PROGRAM MAIN
VAR
	SpeedMotor: MotorVarSpeed_FB;
END_VAR

SpeedMotor(
	Run:= , 
	Direction:= , 
	ConstSpeed:= , 
	Velocity:= , 
	isRunning=> , 
	iActualVel=> );

END_PROGRAM

(* stored: Version 1.1.0.1, ProductVersion 3.1.4024.11
   POU MAIN: Id {af92d42d-f695-4f24-b377-b83b576083d9}, SpecialFunc None *)
